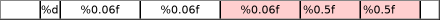
VISUALIZATION _VISU_MarkHistoryEntry  // 440x20
VAR_IN_OUT
	mInst : ST_MarkDefinition;
END_VAR
    Rectangle (220,0 200x20), colour toggle: mInst.sState.bSet
    RoundedRectangle (0,0 40x20), colour variable: mInst.sView.colorFill
    Rectangle (40,0 20x20), "%d", text variable: mInst.nId, colour toggle: mInst.nId=1
    Rectangle (60,0 80x20), "%0.06f", tooltip "square length [mm]", text variable: mInst.fSqLength * 1000
        p4168582468: mInst.fSqLength * 1000
    Rectangle (140,0 80x20), "%0.06f", tooltip "triangle length [mm]", text variable: mInst.fTrLength * 1000
        p4168582468: mInst.fTrLength
    Rectangle (220,0 80x20), "%0.06f", tooltip "detected length [mm]", text variable: mInst.sState.fLengthReal * 1000, colour toggle: mInst.sState.bSet
    Rectangle (300,0 60x20), "%0.5f", text variable: minst.sState.dx * 1000, colour toggle: mInst.sState.bSet
    Rectangle (360,0 60x20), "%0.5f", text variable: minst.sState.dy * 1000, colour toggle: mInst.sState.bSet
    RoundedRectangle (420,0 20x20), tooltip "missed mark", colour toggle: mInst.sState.bMissed, colour variable: mInst.sView.colorFill
END_VISUALIZATION

(* stored: Version 1.1.0.1, ProductVersion 3.1.4024.11
   Visu _VISU_MarkHistoryEntry: Id {1c6fd85b-81a2-4627-9d7d-62e29c4943c7} *)
